// TwinCAT 3 PLC project PLC
// ProgramVersion: 3.1.4024.0
// libraries:
//   Tc2_Standard, * (Beckhoff Automation GmbH)
//   Tc2_System, * (Beckhoff Automation GmbH)
//   Tc2_TcpIp, * (Beckhoff Automation GmbH)
//   Tc2_Utilities, * (Beckhoff Automation GmbH)
//   Tc3_IotBase, * (Beckhoff Automation GmbH)
//   Tc3_JsonXml, * (Beckhoff Automation GmbH)
//   Tc3_Module, * (Beckhoff Automation GmbH)
// project tree:
//   / PlcTask.TcTTO
//   POUs/ DigestTest.TcPOU, JsonSaxHandler_RobotState.TcPOU, MAIN.TcPOU, TcA2B2Kitten.TcPOU, TcA2B2KittenDigest.TcPOU (not stored), UDPTest.TcPOU
// real-time tasks:
//   TASK PlcTask: cycle T#10ms, priority 20, ADS port 350

CONFIGURATION PLC
    RESOURCE PLC ON TwinCAT3
        TASK PlcTask(INTERVAL := T#10ms, PRIORITY := 20);
        PROGRAM MAIN WITH PlcTask : MAIN;
    END_RESOURCE
END_CONFIGURATION

// ---- POUs/MAIN.TcPOU
PROGRAM MAIN
VAR
	myRobot:			TcA2B2Kitten;
	myRobotDigest:		TcA2B2KittenDigest;
	digestTest:			DigestTest;
//	cmdConnect:			BOOL;
//	connectCall:		PLCopenCall;
//	cmdGetRobotState: 	BOOL;
//	getRobotStateCall:	PLCopenCall;
END_VAR


// Call Robot Instance
myRobot();
//myRobotDigest();

//UDPTest();

//digestTest();

(*
/////////////////////////
// Connect

IF cmdConnect THEN
	myRobot.Connect(0, connectCall);
	cmdConnect := FALSE;
END_IF

connectCall();
connectCall.Execute := 0;

// Process command result
IF connectCall.Done THEN
	LogMessage(0, 'Connection Established');
ELSIF connectCall.Error THEN 
	LogMessage(0, 'Connection command error');
ELSIF connectCall.CommandAborted THEN 
	LogMessage(0, 'Connection command aborted');
END_IF

/////////////////////////
// Get Robot State

IF cmdGetRobotState THEN
	myRobot.GetRobotState(getRobotStateCall);
	cmdGetRobotState := FALSE;
END_IF

getRobotStateCall();
getRobotStateCall.Execute := 0;

// Process command result
IF getRobotStateCall.Done THEN
	LogMessage(0, 'GetRobotState Done');
ELSIF getRobotStateCall.Error THEN 
	LogMessage(0, 'GetRobotState command error');
ELSIF getRobotStateCall.CommandAborted THEN 
	LogMessage(0, 'GetRobotState command aborted');
END_IF
*)

END_PROGRAM

// ---- POUs/TcA2B2Kitten.TcPOU
FUNCTION_BLOCK TcA2B2Kitten
VAR_INPUT
END_VAR
VAR_OUTPUT
END_VAR
VAR
	_httpClient:			FB_IotHttpClient;
	_httpRequest:			FB_IotHttpRequest;
	_httpRequestHeader:		FB_IotHttpHeaderFieldMap;
	bTLS:					BOOL;
	bSendGet:				BOOL;
	configureNow:			BOOL;
	requestNow: 			BOOL;
	sContent				: STRING(2000);
	getContentNow: BOOL;
	
	_jsonDomParser : FB_JsonDomParser;
	jsonRoot : SJsonValue;
	jsonProp : SJsonValue;
	parseContentNow: BOOL;
	sState: STRING;
	
	
	_jsonSaxParser : 				FB_JsonSaxReader;
	jsonSaxHandler_RobotState :		JsonSaxHandler_RobotState;
	
	saxParseContentNow: 			BOOL;
END_VAR


IF (NOT _httpClient.bConfigured) OR configureNow THEN 
	//_httpClient.sHostName := '192.168.56.1';
	_httpClient.sHostName := '127.0.0.1';
	_httpClient.nHostPort := 80;
	_httpClient.bKeepAlive := TRUE;
	_httpClient.stTLS.bNoServerCertCheck:=TRUE;
	_httpClient.tConnectionTimeout := T#10S;
	
	IF bTLS THEN
		//_httpClient.stTLS.aPskKey := 0;
		_httpClient.stTLS.bNoServerCertCheck := FALSE;
		//_httpClient.stTLS.nPskKeyLen := 0;
		//_httpClient.stTLS.sCA := '';
		//_httpClient.stTLS.sCert := '';
		_httpClient.stTLS.sCiphers := 'TLS_AES_128_GCM_SHA256';
		//_httpClient.stTLS.sCrl := '';
		//_httpClient.stTLS.sKeyFile := '';
		//_httpClient.stTLS.sKeyPwd := '';
		//_httpClient.stTLS.sPskIdentity := '';
		_httpClient.stTLS.sVersion := 'tlsv1.3';
	END_IF
	configureNow := FALSE;
END_IF

// Method for background communication with the TwinCAT driver. The method must be called cyclically for every client FUB instance.
_httpClient.Execute();

//IF _httpClient.bConnected AND requestNow THEN
IF requestNow AND _httpClient.bConfigured THEN
	//_httpRequest.eCompressionMode := ;
	//_httpRequest.sContentType := ;
	
	_httpRequestHeader.AddField('accept', 'application/xhtml+xml;v=2.0', FALSE);
	_httpRequestHeader.AddField('authorization', 'Basic RGVmYXVsdCBVc2VyOnJvYm90aWNz', FALSE);	// encoded Username: Default User, Password: robotics
	
	_httpRequest.SendRequest(sUri:='/users/rmmp', fbClient:=_httpClient, eRequestType:=ETcIotHttpRequestType.HTTP_Get, pContent:=0, nContentSize:=0, fbHeader:=_httpRequestHeader);
	
	requestNow := FALSE;
END_IF


IF getContentNow THEN
	_httpRequest.GetContent(ADR(sContent), nContentSize:=SIZEOF(sContent), TRUE);
	getContentNow := FALSE;
END_IF


IF parseContentNow THEN
	jsonRoot := _jsonDomParser.ParseDocument(sContent);
	jsonProp := _jsonDomParser.FindMemberPath(jsonRoot, 'state#0/ctrlexecstate');	// See https://infosys.beckhoff.com/english.php?content=../content/1033/tcplclib_tc3_jsonxml/3664369803.html&id=4049129407046606983
	IF (jsonProp <> 0) THEN
  		sState := _jsonDomParser.GetString(jsonProp);
	END_IF
	
	parseContentNow := FALSE; 
END_IF


IF saxParseContentNow THEN
	jsonSaxHandler_RobotState.Reset();
	_jsonSaxParser.Parse(sContent, ipHdl := jsonSaxHandler_RobotState, );
	sState := jsonSaxHandler_RobotState.parsedState;
	
	saxParseContentNow := FALSE; 
END_IF

END_FUNCTION_BLOCK

// ---- POUs/JsonSaxHandler_RobotState.TcPOU
{attribute 'c++_compatible'}
FUNCTION_BLOCK JsonSaxHandler_RobotState IMPLEMENTS ITcJsonSaxHandler
VAR_INPUT
END_VAR
VAR_OUTPUT
	parsedState :	STRING;
END_VAR
VAR
	bStateFound :			BOOL := FALSE;
	bCtrlexecstateFound :	BOOL := FALSE;
END_VAR

(* Example JSON

	{
		"_links": {
			"base": {
				"href": "http://127.0.0.1:80/rw/rapid/"
			},
			"self": {
				"href": "execution"
			}
		},
		"status": {
			"code": 294912
		},
		"state": [
			{
				"_type": "rap-execution",
				"_title": "execution",
				"ctrlexecstate": "stopped",
				"cycle": "forever"
			}
		]
	}

*)

{attribute 'TcTypeSystem'}
{attribute 'no-analysis'}
{attribute 'c++_compatible'}
{attribute 'minimal_input_size' := '4'}
{attribute 'pack_mode' := '4'}
METHOD OnBool : HRESULT
VAR_INPUT
	value	: BOOL;
END_VAR
END_METHOD

{attribute 'TcTypeSystem'}
{attribute 'no-analysis'}
{attribute 'c++_compatible'}
{attribute 'minimal_input_size' := '4'}
{attribute 'pack_mode' := '4'}
METHOD OnDint : HRESULT
VAR_INPUT
	value	: DINT;
END_VAR
END_METHOD

{attribute 'TcTypeSystem'}
{attribute 'no-analysis'}
{attribute 'c++_compatible'}
{attribute 'minimal_input_size' := '4'}
{attribute 'pack_mode' := '4'}
METHOD OnEndArray : HRESULT
VAR_INPUT
	elementCount	: UDINT;
END_VAR
END_METHOD

{attribute 'TcTypeSystem'}
{attribute 'no-analysis'}
{attribute 'c++_compatible'}
{attribute 'minimal_input_size' := '4'}
{attribute 'pack_mode' := '4'}
METHOD OnEndObject : HRESULT
VAR_INPUT
	memberCount	: UDINT;
END_VAR
END_METHOD

{attribute 'TcTypeSystem'}
{attribute 'no-analysis'}
{attribute 'c++_compatible'}
{attribute 'minimal_input_size' := '4'}
{attribute 'pack_mode' := '4'}
METHOD OnKey : HRESULT
VAR_IN_OUT CONSTANT
	key	: STRING;
END_VAR
VAR_INPUT
	len	: UDINT;
END_VAR


IF (key = 'state') THEN
	bStateFound := TRUE;
END_IF

IF bStateFound AND (key = 'ctrlexecstate') THEN
	bCtrlexecstateFound := TRUE;
END_IF
END_METHOD

{attribute 'TcTypeSystem'}
{attribute 'no-analysis'}
{attribute 'c++_compatible'}
{attribute 'minimal_input_size' := '4'}
{attribute 'pack_mode' := '4'}
METHOD OnLint : HRESULT
VAR_INPUT
	value	: LINT;
END_VAR
END_METHOD

{attribute 'TcTypeSystem'}
{attribute 'no-analysis'}
{attribute 'c++_compatible'}
{attribute 'minimal_input_size' := '4'}
{attribute 'pack_mode' := '4'}
METHOD OnLreal : HRESULT
VAR_INPUT
	value	: LREAL;
END_VAR
END_METHOD

{attribute 'TcTypeSystem'}
{attribute 'no-analysis'}
{attribute 'c++_compatible'}
{attribute 'minimal_input_size' := '4'}
{attribute 'pack_mode' := '4'}
METHOD OnNull : HRESULT
END_METHOD

{attribute 'TcTypeSystem'}
{attribute 'no-analysis'}
{attribute 'c++_compatible'}
{attribute 'minimal_input_size' := '4'}
{attribute 'pack_mode' := '4'}
METHOD OnRawNumber : HRESULT
VAR_IN_OUT CONSTANT
	value	: STRING;
END_VAR
VAR_INPUT
	len	: UDINT;
END_VAR
END_METHOD

{attribute 'TcTypeSystem'}
{attribute 'no-analysis'}
{attribute 'c++_compatible'}
{attribute 'minimal_input_size' := '4'}
{attribute 'pack_mode' := '4'}
METHOD OnStartArray : HRESULT
END_METHOD

{attribute 'TcTypeSystem'}
{attribute 'no-analysis'}
{attribute 'c++_compatible'}
{attribute 'minimal_input_size' := '4'}
{attribute 'pack_mode' := '4'}
METHOD OnStartObject : HRESULT
END_METHOD

{attribute 'TcTypeSystem'}
{attribute 'no-analysis'}
{attribute 'c++_compatible'}
{attribute 'minimal_input_size' := '4'}
{attribute 'pack_mode' := '4'}
METHOD OnString : HRESULT
VAR_IN_OUT CONSTANT
	value	: STRING;
END_VAR
VAR_INPUT
	len	: UDINT;
END_VAR

IF bCtrlexecstateFound THEN
	parsedState := value;
	OnString := S_FALSE;
END_IF
END_METHOD

{attribute 'TcTypeSystem'}
{attribute 'no-analysis'}
{attribute 'c++_compatible'}
{attribute 'minimal_input_size' := '4'}
{attribute 'pack_mode' := '4'}
METHOD OnUdint : HRESULT
VAR_INPUT
	value	: UDINT;
END_VAR
END_METHOD

{attribute 'TcTypeSystem'}
{attribute 'no-analysis'}
{attribute 'c++_compatible'}
{attribute 'minimal_input_size' := '4'}
{attribute 'pack_mode' := '4'}
METHOD OnUlint : HRESULT
VAR_INPUT
	value	: ULINT;
END_VAR
END_METHOD

METHOD Reset : bool
VAR_INPUT
END_VAR

VAR
	bStateFound: BOOL;
END_VAR

// Reset parsing state variables
bStateFound := FALSE;
bCtrlexecstateFound := FALSE;
END_METHOD

{attribute 'TcTypeSystem'}
{attribute 'no-analysis'}
{attribute 'c++_compatible'}
{attribute 'minimal_input_size' := '4'}
{attribute 'pack_mode' := '4'}
METHOD TcAddRef : UDINT
END_METHOD

{attribute 'TcTypeSystem'}
{attribute 'no-analysis'}
{attribute 'c++_compatible'}
{attribute 'minimal_input_size' := '4'}
{attribute 'pack_mode' := '4'}
METHOD TcQueryInterface : HRESULT
VAR_INPUT
	iid	: REFERENCE TO IID;
	pipItf	: POINTER TO PVOID;
END_VAR
END_METHOD

{attribute 'TcTypeSystem'}
{attribute 'no-analysis'}
{attribute 'c++_compatible'}
{attribute 'minimal_input_size' := '4'}
{attribute 'pack_mode' := '4'}
METHOD TcRelease : UDINT
END_METHOD

END_FUNCTION_BLOCK

// ---- POUs/DigestTest.TcPOU
FUNCTION_BLOCK DigestTest
VAR_INPUT
END_VAR
VAR_OUTPUT
END_VAR
VAR
	un : STRING;
	pw : STRING;
	realm : STRING;
	meth : STRING;
	uri : STRING;
	qop : STRING;
	nonce : STRING;
	cnonce : STRING;
	nc : STRING;
	
	tempString : STRING(1000);
	
	retVal: BOOL;
	
	h1_byArr: ARRAY[0..15] OF BYTE;
	h1_hexStr: STRING;
	h2_byArr: ARRAY[0..15] OF BYTE;
	h2_hexStr: STRING;
	response_byArr: ARRAY[0..15] OF BYTE;
	response_hexStr: STRING;
	
	calculateNow : BOOL;
	i: INT;
END_VAR



IF calculateNow THEN
	
	// Values collected via wireshark
	un := 'Default User';
	pw := 'robotics';
	realm := 'validusers@robapi.abb';
	meth := 'GET';
	uri := '/rw/rapid/execution';
	qop := 'auth';
	nonce := 'MGY0Yjc2MGY2Y2QyZjAwNzp2YWxpZHVzZXJzQHJvYmFwaS5hYmI6MTkwMjg5NjRlNGE6MA==';
	cnonce := 'diddLOPR';
	nc := '00000001';
	
	
	tempString := '';
	tempString := CONCAT(tempString, un);
	tempString := CONCAT(tempString, ':');
	tempString := CONCAT(tempString, realm);
	tempString := CONCAT(tempString, ':');
	tempString := CONCAT(tempString, pw);
	
	retVal := F_GenerateHashValue(E_HashMode.HASH_MD5, ADR(tempString), LEN(tempString), ADR(h1_byArr), SIZEOF(h1_byArr));
	
	//h1_hexStr := DATA_TO_HEXSTR(ADR(h1_byArr), SIZEOF(h1_byArr), TRUE); // this method adds unnecessary space characters between bytes
	h1_hexStr := '';
	FOR i := 0 TO 15 DO
		h1_hexStr := CONCAT(h1_hexStr, BYTE_TO_HEXSTR(h1_byArr[i], 2, TRUE));
	END_FOR
	// expected value: 952890790eb23290847e6f4d57e76d86
	
	
	tempString := '';
	tempString := CONCAT(tempString, meth);
	tempString := CONCAT(tempString, ':');
	tempString := CONCAT(tempString, uri);
	
	retVal := F_GenerateHashValue(E_HashMode.HASH_MD5, ADR(tempString), LEN(tempString), ADR(h2_byArr), SIZEOF(h2_byArr));
	
	h2_hexStr := '';
	FOR i := 0 TO 15 DO
		h2_hexStr := CONCAT(h2_hexStr, BYTE_TO_HEXSTR(h2_byArr[i], 2, TRUE));
	END_FOR
	// expected value: 30bb6c0952d8c10cb9b2240a3772c67b
	
	
	tempString := '';
	tempString := CONCAT(tempString, h1_hexStr);
	tempString := CONCAT(tempString, ':');
	tempString := CONCAT(tempString, nonce);
	tempString := CONCAT(tempString, ':');
	tempString := CONCAT(tempString, nc);
	tempString := CONCAT(tempString, ':');
	tempString := CONCAT(tempString, cnonce);
	tempString := CONCAT(tempString, ':');
	tempString := CONCAT(tempString, qop);
	tempString := CONCAT(tempString, ':');
	tempString := CONCAT(tempString, h2_hexStr);
	
	retVal := F_GenerateHashValue(E_HashMode.HASH_MD5, ADR(tempString), LEN(tempString), ADR(response_byArr), SIZEOF(response_byArr));
	
	response_hexStr := '';
	FOR i := 0 TO 15 DO
		response_hexStr := CONCAT(response_hexStr, BYTE_TO_HEXSTR(response_byArr[i], 2, TRUE));
	END_FOR
	// expected value: c36e30cdd2961584cd41f6f49f6bcbba
	
	
	
	calculateNow := FALSE;
END_IF

END_FUNCTION_BLOCK

// ---- POUs/UDPTest.TcPOU
PROGRAM UDPTest
VAR
	socketCreate:	FB_SocketUdpCreate;
	socketSend:		FB_SocketUdpSendTo;
	createNow: 		BOOL;
	sendNow:		BOOL;
	sMsg:			STRING[20] := 'Hello World';
	configCreate: 	BOOL := true;
	configSend: 	BOOL := TRUE;
END_VAR




IF configCreate THEN
	socketCreate.sSrvNetId := '';
	socketCreate.sLocalHost := '127.0.0.1';
	socketCreate.nLocalPort := 52123;
	socketCreate.tTimeout := T#5S;
	configCreate := FALSE;
END_IF


//IF createNow THEN
	socketCreate.bExecute := createNow;
//	createNow := FALSE;
//END_IF

IF configSend THEN
	socketSend.sSrvNetId := '';
	socketSend.sRemoteHost := '127.0.0.1';
	socketSend.nRemotePort := 8000;
	socketSend.cbLen := LEN(sMsg);
	socketSend.pSrc := ADR(sMsg);
	socketSend.tTimeout := T#5S;
	configSend := FALSE;
END_IF

socketSend.hSocket := socketCreate.hSocket;

socketSend.bExecute := sendNow;
sendNow := FALSE;

// Call fbs
socketCreate();
socketSend();

END_PROGRAM
